{attribute 'qualified_only'}
VAR_GLOBAL
	bsSensor		: BOOL; //s sensor for detection cylinder NO
	bM2Spindisk		:BOOL; // spins disk Motor
	bM1Motor		:BOOL; // M1 motor 
	
END_VAR

(* stored: Version 1.1.0.1, ProductVersion 3.1.4024.12
   GVL input: Id {20c0a195-e80f-4f04-a815-7ab5ea192169} *)
